ABB RobotStudio station: Session6.rspag

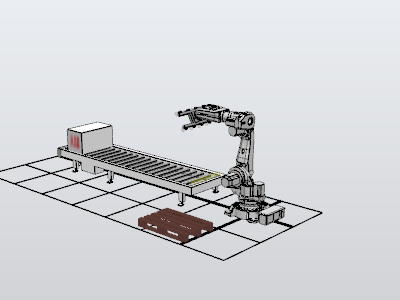
--- station ---
Station Session6d (saved by RobotStudio 24.2.10821.1)
Controller IRB6620_SC_system
  mechanical unit ROB_1: IRB6620_150_220__01_2, 6 joints, base frame (0, 0, 0) mm
Layout (positions relative to the parent item):
  - IRB6620_150_220__01_2 [mechanism, from %ABB.RobotStudio.Models.IRB6620%\IRB6620_150_220_G_01.rslib] at (0, 0, 0) mm; joint values [0, 0, 0, 0, 0.5236, 0] (rad or m)
  - SC_VacuumGripper [smart component, from Libraries\SC_VacuumGripper.rslib] at (1380.21, 0, 1755) mm, rotated rx 180 ry 60 rz 180 deg
      properties: PartInGripper=(none)
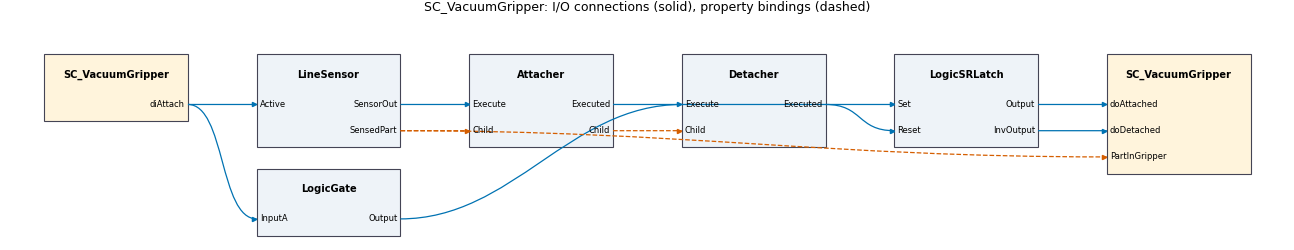
      connections:
        SC_VacuumGripper.diAttach -> LineSensor.Active
        LineSensor.SensorOut -> Attacher.Execute
        SC_VacuumGripper.diAttach -> LogicGate.InputA
        LogicGate.Output -> Detacher.Execute
        Attacher.Executed -> LogicSRLatch.Set
        Detacher.Executed -> LogicSRLatch.Reset
        LogicSRLatch.Output -> SC_VacuumGripper.doAttached
        LogicSRLatch.InvOutput -> SC_VacuumGripper.doDetached
        LineSensor.SensedPart => Attacher.Child
        Attacher.Child => Detacher.Child
        LineSensor.SensedPart => SC_VacuumGripper.PartInGripper
    - VacuumGripper [mechanism, from Libraries\SC_VacuumGripper.rslib] at (0, 0, 0) mm
    - LineSensor [smart component, from Components\LineSensor.rslib]
        properties: Start=[0 0 0.15]; End=[0 0 0.25]; Length=0.1; Radius=0.001; Tag=(none); SensedPart=(none); SensedPoint=[0 0 0]
      - _sensorPart_ [part, from Libraries\SC_VacuumGripper.rslib]
    - Attacher [smart component, from Components\Attacher.rslib]
        properties: Parent=VacuumGripper; Flange=0; Child=(none); Mount=false; Offset=[0 0 0]; Orientation=[0 0 0]
    - Detacher [smart component, from Components\Detacher.rslib]
        properties: Child=(none); KeepPosition=true
    - LogicGate [smart component, from Components\LogicGate.rslib]
        properties: Operator=NOT; Delay=0
    - LogicSRLatch [smart component, from Components\LogicSRLatch.rslib]
  - SC_InFeeder [smart component, from Libraries\SC_InFeeder2.rslib]
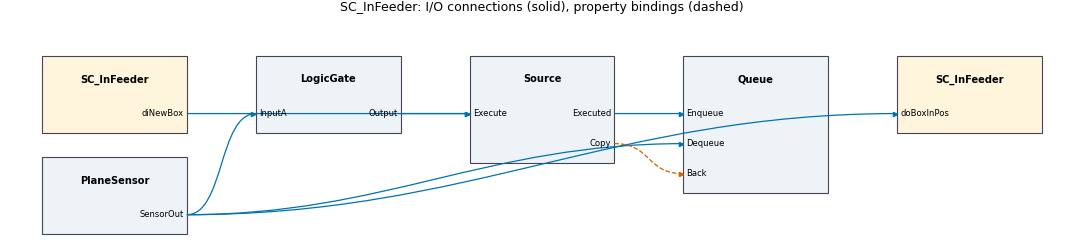
      connections:
        SC_InFeeder.diNewBox -> Source.Execute
        Source.Executed -> Queue.Enqueue
        PlaneSensor.SensorOut -> Queue.Dequeue
        PlaneSensor.SensorOut -> SC_InFeeder.doBoxInPos
        PlaneSensor.SensorOut -> LogicGate.InputA
        LogicGate.Output -> Source.Execute
        Source.Copy => Queue.Back
    - InFeeder [part, from Libraries\SC_InFeeder2.rslib]
    - Source [smart component, from Components\Source.rslib]
        properties: Source=box; Copy=(none); Parent=(none); Position=[0 0 0]; Orientation=[0 0 0]; Transient=false; PhysicsBehavior=-1
    - LinearMover [smart component, from Components\LinearMover.rslib]
        properties: Object=Queue; Direction=[-1 0 0]; Speed=0.5; Reference=Global; ReferenceObject=(none)
    - Queue [smart component, from Components\Queue.rslib]
        properties: Back=(none); Front=(none); Queue={cc8bc1f8-4511-4c9a-9a84-cfeea6807d22}; NumberOfObjects=1
    - PlaneSensor [smart component, from Components\PlaneSensor.rslib]
        properties: Origin=[1.14 0.485 0.445]; Axis1=[0 0 0.1]; Axis2=[0 -0.93 0]; Tag=(none); SensedPart=(none)
      - _sensorPart_ [part, from Libraries\SC_InFeeder2.rslib]
    - LogicGate [smart component, from Components\LogicGate.rslib]
        properties: Operator=NOT; Delay=0
  - SC_OutPallet [smart component, from Libraries\SC_OutPallet2.rslib]
      properties: PartFromRobot=(none)
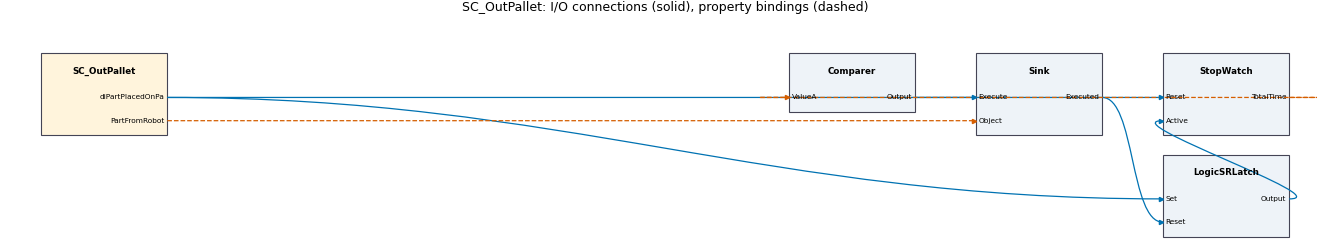
      connections:
        SC_OutPallet.diPartPlacedOnPallet -> StopWatch.Reset
        SC_OutPallet.diPartPlacedOnPallet -> LogicSRLatch.Set
        LogicSRLatch.Output -> StopWatch.Active
        Comparer.Output -> Sink.Execute
        Sink.Executed -> LogicSRLatch.Reset
        SC_OutPallet.PartFromRobot => Sink.Object
        StopWatch.TotalTime => Comparer.ValueA
    - Euro Pallet [graphiccomponentgroup, from Libraries\SC_OutPallet2.rslib] at (0, 1100, 0) mm
      - Body 1 [part, from Libraries\SC_OutPallet2.rslib]
    - Sink [smart component, from Components\Sink.rslib]
        properties: Object=(none)
    - Comparer [smart component, from Components\Comparer.rslib]
        properties: ValueA=0; Operator=>=; ValueB=2
    - StopWatch [smart component, from Components\StopWatch.rslib]
        properties: TotalTime=0; LapTime=0; AutoReset=false
    - LogicSRLatch [smart component, from Components\LogicSRLatch.rslib]
  - box [part, from Library\box.rslib]
Attachment: SC_VacuumGripper is attached to IRB6620_150_220__01_2 / Link6
Station logic (signal -> signal, property => property):
  SC_VacuumGripper.doDetached -> SC_OutPallet.diPartPlacedOnPallet
  IRB6620_SC_system.doNewBox -> SC_InFeeder.diNewBox
  SC_InFeeder.doBoxInPos -> IRB6620_SC_system.diBoxInPos
  IRB6620_SC_system.doVacuum -> SC_VacuumGripper.diAttach
  SC_VacuumGripper.doAttached -> IRB6620_SC_system.diVacuum
  SC_VacuumGripper.PartInGripper => SC_OutPallet.PartFromRobot

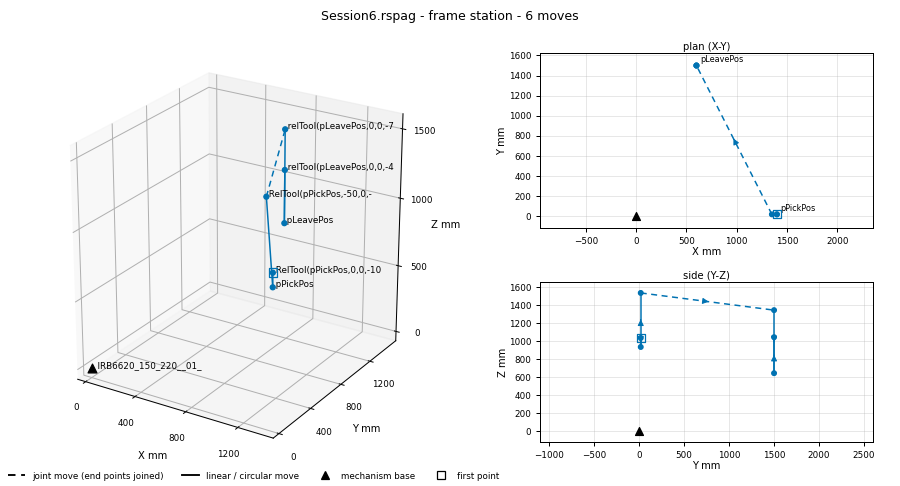
[picture p0: tool path of Session6.rspag in frame station, 6 of 6 moves have a stored position in this frame; points joined in program order, loops and branches not executed]
--- Backups/IRB6620_SC_system/RAPID/TASK1/PROGMOD/CalibData.mod ---
MODULE CalibData
	TASK PERS wobjdata wobjInFeeder:=[FALSE,TRUE,"",[[1080,-535,435],[1,0,0,0]],[[0,0,0],[1,0,0,0]]];
	TASK PERS wobjdata wobOutPallet:=[FALSE,TRUE,"",[[0,1100,144],[1,0,0,0]],[[0,0,0],[1,0,0,0]]];
	PERS tooldata tGripper:=[TRUE,[[0,0,197.5],[1,0,0,0]],[25,[0,0.00109327,116.889],[1,0,0,0],0,0,0]];
ENDMODULE

--- Backups/IRB6620_SC_system/RAPID/TASK1/PROGMOD/modCalibData.mod ---
%%%
   VERSION: 1
   LANGUAGE: ENGLISH
%%%

MODULE modCalibData

ENDMODULE

--- Backups/IRB6620_SC_system/RAPID/TASK1/PROGMOD/modRobotStudio.mod ---
MODULE modRobotStudio
    CONST robtarget pPickPos:=[[320,555,500],[0,1,0,0],[0,0,0,0],[9E9,9E9,9E9,9E9,9E9,9E9]];
    CONST robtarget pLeavePos:=[[600,400,500],[0,0.707106781,0.707106781,0],[0,0,0,0],[9E9,9E9,9E9,9E9,9E9,9E9]];
    CONST robtarget Target_10:=[[1400.00000000001,20,835],[8.32667268468867E-16,0,1,0],[0,0,0,0],[9E9,9E9,9E9,9E9,9E9,9E9]];

    PROC PickLeave()
        MoveJ RelTool(pPickPos,0,0,-100),v1000,z10,tGripper\WObj:=wobjInFeeder;
        WaitDI diBoxInPos,1;
        MoveL pPickPos,v100,fine,tGripper\WObj:=wobjInFeeder;
        SetDO doVacuum,1;
        WaitDI diVacuum,1;
        MoveL RelTool(pPickPos,-50,0,-600),v1000,z10,tGripper\WObj:=wobjInFeeder;
        MoveJ relTool(pLeavePos,0,0,-700),v1000,z10,tGripper\WObj:=wobOutPallet;
        MoveL pLeavePos,v1000,fine,tGripper\WObj:=wobOutPallet;
        SetDO doVacuum,0;
        WaitDI diVacuum,0;
        MoveL relTool(pLeavePos,0,0,-400),v1000,z10,tGripper\WObj:=wobOutPallet;
    ENDPROC


    PROC main()
        SetDO doVacuum,0;
        WaitDI diVacuum,0;
        PulseDO doNewBox;
        WHILE TRUE DO
            PickLeave;
        ENDWHILE
    ENDPROC
ENDMODULE

--- Backups/IRB6620_SC_system/RAPID/TASK1/SYSMOD/LINKEDM.sys ---
%%%
  VERSION:1
  LANGUAGE:ENGLISH
%%%

MODULE LINKEDM (SYSMODULE)

! FOLLOWER
!     Name of electronically linked follower axis used by operator at teach pendent.
      PERS string l_f_axis_name{5}       :=  ["",  "", "", "", ""];

!     Name of the mechanical unit for follower axis.
      PERS string l_f_mecunt_n{5}  :=  ["", "", "", "", ""];

!     Linked follower axis number in the mechanical unit (first axis in mech. unit is number 1).
      PERS num l_f_axis_no{5}      :=  [0,          0,   0,  0,  0];

! MASTER
!     Name of the mechanical unit for linked master axis.
      PERS string l_m_mecunt_n{5} :=  ["", "", "", "", ""];

!     Linked master axis number in the mechanical unit (first axis in mech. unit is number 1).
!     See axis number table in documentation for different master mechanical units.
      PERS num l_m_axis_no{5}     :=  [0,  0,  0,  0,  0];

! POSITION OFFSET
!     The increase of the allowed offset position between the master and follower
!     positions, used when starting AUTO mode. As soon as the offset is decreased
!     the old configurated parameter is used.
!     Example: 3 => the configurated value of allowed offset is increased 3 times.
      PERS num offset_ratio{5}       :=  [10,  10,   10,  10,  10];

! SPEED RATIO
!     Speed_ratio used in AUTO and JOG modes [ very_slow   slow    normal    fast]
!     Value 1 = max allowed manual speed.
      CONST num speed_ratio {20}      := [0.01, 0.01, 0.01, 0.01, 0.01,
                                          0.05, 0.05, 0.05, 0.05, 0.05,
                                          0.20, 0.20, 0.20, 0.20, 0.20,
                                          1.00, 1.00, 1.00, 1.00, 1.00];

! STEP SIZE
!     Displacement position used in JOG mode for each activation of positive or
!     negative movement.                  [very_short    short   normal   long]
!     Unit degees or meter.
      CONST num displacement {20}     := [0.001, 0.001, 0.001, 0.001, 0.001,
                                          0.005, 0.005, 0.005, 0.005, 0.005,
                                          0.020, 0.020, 0.020, 0.020, 0.020,
                                          0.100, 0.100, 0.100, 0.100, 0.100];


!-------------------------------------------------------------
 PROC Linked_m ()
      Linked_m_exe ;
 ENDPROC
ENDMODULE

--- Backups/IRB6620_SC_system/SYSPAR/EIO.cfg ---
EIO:CFG_1.0:6:1::
#
EIO_SIGNAL:

      -Name "diBoxInPos" -SignalType "DI" -Access "All"

      -Name "diVacuum" -SignalType "DI" -Access "All"

      -Name "doNewBox" -SignalType "DO" -Access "All"

      -Name "doVacuum" -SignalType "DO" -Access "All"
